{attribute addProperty BoxType "EK1122-0000-0018"}
{attribute addProperty Id "Beckhoff_EL67xxsub_EK1100EK1100_179A0949162"}
{attribute addProperty CRC "1864869311"}
{attribute addProperty SizeInBites "16"}
{attribute addProperty SizeInBytes "2"}
TYPE Beckhoff_EL67xxEK1122_6F27A5BF EXTENDS EK1122_179A0949 :
STRUCT
	{attribute addProperty Name "Beckhoff_EL67xxsub_EK1100"}
	Beckhoff_EL67xxsub_EK1100 : EK1100_179A0949;
END_STRUCT
END_TYPE

(* stored: Version 1.2.0.0, ProductVersion 3.1.4024.9
   DUT Beckhoff_EL67xxEK1122_6F27A5BF: Id {64fdc73a-83ec-4eb2-96e0-ac7b0085db59} *)
